(* PLC project servo_control, Dassault Systèmes ControlBuild 2024x *)
(* stored: creationDateTime 2023-10-04T11:03:55-01:00 *)

(* This module control the accesses to control the motion drive *)
FUNCTION_BLOCK motion_control.servo_control
  VAR_INPUT
    HomeCmd : BOOL := false;
    MoveVelCmd : BOOL := false;
    MoveAbsCmd : BOOL := false;
    MoveVel1ManualCmd : BOOL := false;
    MoveVel2ManualCmd : BOOL := false;
    MoveAbs1ManualCmd : BOOL := false;
    MoveAbs2ManualCmd : BOOL := false;
    StopCmd : BOOL := false;
    MovePosition : REAL := 0.0;
    MoveSpeed : REAL := 100.0;
    MoveAcceleration : REAL := 100.0;
    MoveDeceleration : REAL := 100.0;
    offsetAxToMa : REAL := 0.0;
  END_VAR
  VAR_INPUT
    physicalPosInit : REAL := 0.0;
    MAX_SPEED : REAL(0.0..3.4e+38) := 1000.0;
  END_VAR
  VAR_IN_OUT
    status : INT := 0;
    errorFlag : INT := 0;
    IOActualPositionAx : REAL := 0.0;
    IOVelDone : BOOL := false;
    IOAbsDone : BOOL := false;
    IOActualVelocity : REAL := 0.0;
  END_VAR
  VAR_OUTPUT
    OperationMode : INT := 0;
  END_VAR
  VAR_OUTPUT
    StatusReady : BOOL := true;
    StatusMove : BOOL := false;
    StatusStand : BOOL := false;
    ActualPositionMa : REAL := 0.0;
    ActualVelocity : REAL := 0.0;
    MaximumVelocity : REAL := 0.0;
  END_VAR
  VAR_OUTPUT
    VelEnabled : BOOL := false;
    VelCmd : BOOL := false;
    PosEnabled : BOOL := false;
    PosCmd : BOOL := false;
    Position : REAL := 0.0;
    Speed : REAL := 0.0;
  END_VAR
  VAR
    ManualMode : INT := 0;
    initDone : BOOL := false;
    ActualPositionMa1 : REAL := 0.0;
    offsetAxToMa1 : REAL := 0.0;
  END_VAR
  VAR CONSTANT
    HOME_POSITION : REAL := 100.0;
    MANUAL_POSITION1 : REAL := 0.0;
    MANUAL_POSITION2 : REAL := 150.0;
    MANUAL_SPEED1 : REAL := -100.0;
    MANUAL_SPEED2 : REAL := 100.0;
    MANUAL_SPEED : REAL := 100.0;
  END_VAR


ACTION C_source_code:
/* ----------------------------------------------------------------	*/
/* Type : Model of Operative Behaviour					*/
/* Category :  motion control						*/
/* Author : 									*/
/* Update date : June 2021							*/
/* ----------------------------------------------------------------	*/
/* This module control the accesses to control the motion drive 	*/
/* ----------------------------------------------------------------	*/

if (initDone == 0) {
	IOActualPositionAx = physicalPosInit;
}
// modification of ref position
if (offsetAxToMa != offsetAxToMa1) {
	ActualPositionMa += (offsetAxToMa - offsetAxToMa1);
	ActualPositionMa1 += (offsetAxToMa - offsetAxToMa1);
}
if (MoveVel1ManualCmd && StatusReady) {
	ManualMode = 1;
	StatusReady = 0;
	Speed = MANUAL_SPEED1;
	PosEnabled = 0;
	VelEnabled = 1;
	PosCmd = 0;
	VelCmd = 1;
}
if (MoveVel2ManualCmd && StatusReady) {
	ManualMode = 1;
	StatusReady = 0;
	Speed = MANUAL_SPEED2;
	PosEnabled = 0;
	VelEnabled = 1;
	PosCmd = 0;
	VelCmd = 1;
}
if (MoveAbs1ManualCmd && StatusReady) {
	ManualMode = 3;
	StatusReady = 0;
	Position = MANUAL_POSITION1;
	Speed = MANUAL_SPEED;
	PosEnabled = 1;
	VelEnabled = 0;
	PosCmd = 1;
	VelCmd = 0;
}
if (MoveAbs2ManualCmd && StatusReady) {
	ManualMode = 3;
	StatusReady = 0;
	Position = MANUAL_POSITION2;
	Speed = MANUAL_SPEED;
	PosEnabled = 1;
	VelEnabled = 0;
	PosCmd = 1;
	VelCmd = 0;
}
if (HomeCmd && StatusReady) {
	OperationMode = 1;
	StatusReady = 0;
	Position = HOME_POSITION;
	Speed = MoveSpeed;
	PosEnabled = 1;
	VelEnabled = 0;
	PosCmd = 1;
	VelCmd = 0;
}
if (MoveVelCmd && StatusReady) {
	OperationMode = 2;
	StatusReady = 0;
	Speed = MoveSpeed;
	PosEnabled = 0;
	VelEnabled = 1;
	PosCmd = 0;
	VelCmd = 1;
}
if (MoveAbsCmd && StatusReady) {
	OperationMode = 3;
	StatusReady = 0;
	Position = MovePosition - offsetAxToMa;
	Speed = MoveSpeed;
	PosEnabled = 1;
	VelEnabled = 0;
	PosCmd = 1;
	VelCmd = 0;
}
if ((OperationMode != 0 && StopCmd) || (OperationMode == 2 && !MoveVelCmd) || status == 5) {
	OperationMode = 0;
	ManualMode = 0;
	PosCmd = 0;
	VelCmd = 0;
}
if (ManualMode == 1 && !MoveVel1ManualCmd && !MoveVel2ManualCmd) {
	OperationMode = 0;
	ManualMode = 0;
	PosCmd = 0;
	VelCmd = 0;
}
if (OperationMode == 0 && ManualMode == 0 && status == 0) {
	StatusReady = 1;
	PosEnabled = 0;
	VelEnabled = 0;
}

ActualVelocity = IOActualVelocity;
StatusMove = (ActualVelocity != 0.0);
StatusStand = (ActualVelocity == 0.0);
ActualPositionMa1 = ActualPositionMa;
ActualPositionMa = IOActualPositionAx + offsetAxToMa;
offsetAxToMa1 = offsetAxToMa;
MaximumVelocity = MAX_SPEED;

initDone = 1;
END_ACTION
END_FUNCTION_BLOCK
